(*$
	Returns <i>jog_activation_condition</i> of the instance <b><i>this</i></b>.
$*)
FUNCTION jog_manager_get_jog_activation_condition : BOOL
VAR_IN_OUT
    CONVERSION_this:	jog_manager;	(*$ Instance to which the method applies $*)
END_VAR

jog_manager_get_jog_activation_condition := CONVERSION_this.jog_activation_condition;

END_FUNCTION

(* stored: Version 1.1.0.1, ProductVersion 3.1.4022.12
   POU jog_manager_get_jog_activation_condition: Id {262d18cd-28fc-4b6a-babe-153701acee53}, SpecialFunc None *)
